FUNCTION_BLOCK FB_System_MVWW_Ablaufsteuerung
VAR_IN_OUT
	Zustand					: ST_System_MVWW_Zustand;
	Stellwert				: ST_System_MVWW_Stellwert;
	Steuerung				: ST_System_MVWW_Steuerung;
END_VAR
VAR_INPUT
	Zustand_Stellventil		: ST_SV_Zustand;
	Zustand_Pumpe			: ST_PU_Zustand;
END_VAR
VAR_OUTPUT
END_VAR
VAR
END_VAR

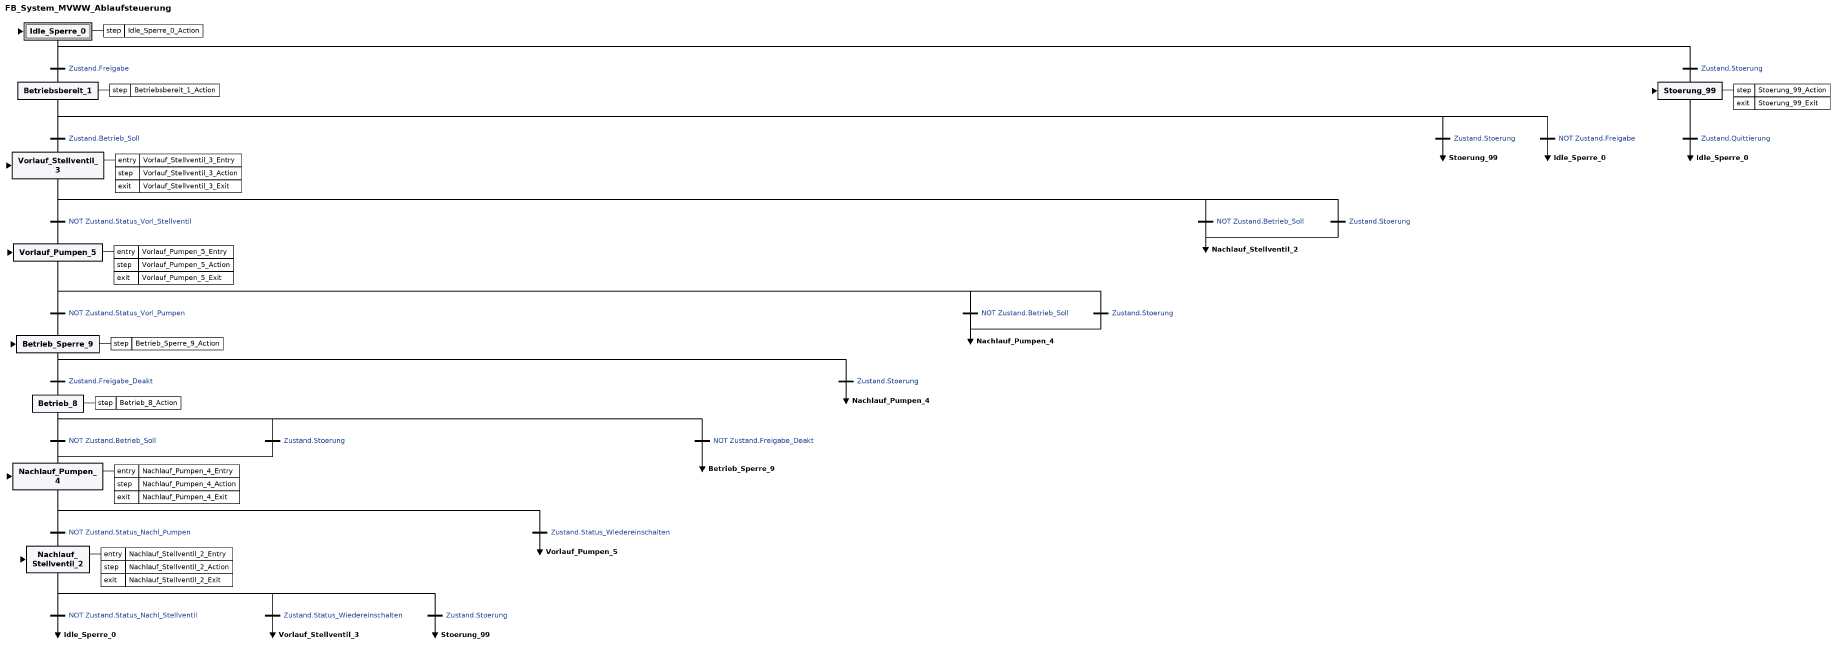
INITIAL_STEP Idle_Sperre_0:
    Idle_Sperre_0_Action(N);  // step action
END_STEP
TRANSITION FROM Idle_Sperre_0 TO Betriebsbereit_1
    := Zustand.Freigabe;
END_TRANSITION
TRANSITION FROM Idle_Sperre_0 TO Stoerung_99
    := Zustand.Stoerung;
END_TRANSITION
STEP Stoerung_99:
    Stoerung_99_Action(N);  // step action
    Stoerung_99_Exit(P0);  // exit action
END_STEP
TRANSITION FROM Stoerung_99 TO Idle_Sperre_0
    := Zustand.Quittierung;
END_TRANSITION
STEP Betriebsbereit_1:
    Betriebsbereit_1_Action(N);  // step action
END_STEP
TRANSITION FROM Betriebsbereit_1 TO Vorlauf_Stellventil_3
    := Zustand.Betrieb_Soll;
END_TRANSITION
TRANSITION FROM Betriebsbereit_1 TO Stoerung_99
    := Zustand.Stoerung;
END_TRANSITION
TRANSITION FROM Betriebsbereit_1 TO Idle_Sperre_0
    := NOT Zustand.Freigabe;
END_TRANSITION
STEP Vorlauf_Stellventil_3:
    Vorlauf_Stellventil_3_Entry(P1);  // entry action
    Vorlauf_Stellventil_3_Action(N);  // step action
    Vorlauf_Stellventil_3_Exit(P0);  // exit action
END_STEP
TRANSITION FROM Vorlauf_Stellventil_3 TO Vorlauf_Pumpen_5
    := NOT Zustand.Status_Vorl_Stellventil;
END_TRANSITION
TRANSITION FROM Vorlauf_Stellventil_3 TO Nachlauf_Stellventil_2
    := NOT Zustand.Betrieb_Soll;
END_TRANSITION
TRANSITION FROM Vorlauf_Stellventil_3 TO Nachlauf_Stellventil_2
    := Zustand.Stoerung;
END_TRANSITION
STEP Vorlauf_Pumpen_5:
    Vorlauf_Pumpen_5_Entry(P1);  // entry action
    Vorlauf_Pumpen_5_Action(N);  // step action
    Vorlauf_Pumpen_5_Exit(P0);  // exit action
END_STEP
TRANSITION FROM Vorlauf_Pumpen_5 TO Betrieb_Sperre_9
    := NOT Zustand.Status_Vorl_Pumpen;
END_TRANSITION
TRANSITION FROM Vorlauf_Pumpen_5 TO Nachlauf_Pumpen_4
    := NOT Zustand.Betrieb_Soll;
END_TRANSITION
TRANSITION FROM Vorlauf_Pumpen_5 TO Nachlauf_Pumpen_4
    := Zustand.Stoerung;
END_TRANSITION
STEP Betrieb_Sperre_9:
    Betrieb_Sperre_9_Action(N);  // step action
END_STEP
TRANSITION FROM Betrieb_Sperre_9 TO Betrieb_8
    := Zustand.Freigabe_Deakt;
END_TRANSITION
TRANSITION FROM Betrieb_Sperre_9 TO Nachlauf_Pumpen_4
    := Zustand.Stoerung;
END_TRANSITION
STEP Betrieb_8:
    Betrieb_8_Action(N);  // step action
END_STEP
TRANSITION FROM Betrieb_8 TO Nachlauf_Pumpen_4
    := NOT Zustand.Betrieb_Soll;
END_TRANSITION
TRANSITION FROM Betrieb_8 TO Nachlauf_Pumpen_4
    := Zustand.Stoerung;
END_TRANSITION
TRANSITION FROM Betrieb_8 TO Betrieb_Sperre_9
    := NOT Zustand.Freigabe_Deakt;
END_TRANSITION
STEP Nachlauf_Pumpen_4:
    Nachlauf_Pumpen_4_Entry(P1);  // entry action
    Nachlauf_Pumpen_4_Action(N);  // step action
    Nachlauf_Pumpen_4_Exit(P0);  // exit action
END_STEP
TRANSITION FROM Nachlauf_Pumpen_4 TO Nachlauf_Stellventil_2
    := NOT Zustand.Status_Nachl_Pumpen;
END_TRANSITION
TRANSITION FROM Nachlauf_Pumpen_4 TO Vorlauf_Pumpen_5
    := Zustand.Status_Wiedereinschalten;
END_TRANSITION
STEP Nachlauf_Stellventil_2:
    Nachlauf_Stellventil_2_Entry(P1);  // entry action
    Nachlauf_Stellventil_2_Action(N);  // step action
    Nachlauf_Stellventil_2_Exit(P0);  // exit action
END_STEP
TRANSITION FROM Nachlauf_Stellventil_2 TO Idle_Sperre_0
    := NOT Zustand.Status_Nachl_Stellventil;
END_TRANSITION
TRANSITION FROM Nachlauf_Stellventil_2 TO Vorlauf_Stellventil_3
    := Zustand.Status_Wiedereinschalten;
END_TRANSITION
TRANSITION FROM Nachlauf_Stellventil_2 TO Stoerung_99
    := Zustand.Stoerung;
END_TRANSITION

ACTION Betrieb_8_Action:
(* Stellwert setzen *)
Stellwert.Anford_Stellventil	:= TRUE;
Stellwert.Anford_Pumpe			:= TRUE;

(* Zustand setzen *)
Zustand.Status					:= E_System_MVWW_Zustand_Status_Betrieb;
END_ACTION

ACTION Betrieb_Sperre_9_Action:
(* Stellwert setzen *)
Stellwert.Anford_Stellventil		:= TRUE;
Stellwert.Anford_Pumpe				:= TRUE;


(* Zustand setzen *)
Zustand.Status						:= E_System_MVWW_Zustand_Status_Betrieb_Sperre;
END_ACTION

ACTION Betriebsbereit_1_Action:
(* Stellwert setzen *)
Stellwert.Anford_Stellventil	:= FALSE;
Stellwert.Anford_Pumpe			:= FALSE;

(* Zustand setzen *)
Zustand.Status			:= E_System_MVWW_Zustand_Status_Betriebsbereit;
END_ACTION

ACTION Idle_Sperre_0_Action:
(* Stellwert setzen *)
Stellwert.Anford_Stellventil		:= FALSE;
Stellwert.Anford_Pumpe				:= FALSE;

(* Zustand setzen *)
Zustand.Status						:= E_System_MVWW_Zustand_Status_Idle_Sperre;

(* Quittierungszustand auf False setzen, damit das System bei einer erneuten Störung nicht direkt wieder angeschaltet wird *)
Steuerung.Quittierung				:= FALSE;
END_ACTION

ACTION Nachlauf_Pumpen_4_Action:
(* Stellwert setzen *)
Stellwert.Anford_Stellventil	:= FALSE;
Stellwert.Anford_Pumpe			:= FALSE;


(* Zustand setzen *)
Zustand.Status						:= E_System_MVWW_Zustand_Status_Nachl_Pumpe;
Zustand.Status_Nachl_Pumpen			:= Zustand_Pumpe.Betrieb OR  Zustand_Pumpe.Status_Nachl;
Zustand.Status_Wiedereinschalten 	:= Zustand.Betrieb_Soll AND Stellwert.Einschalten;
END_ACTION

ACTION Nachlauf_Pumpen_4_Entry:
Zustand.Status_Nachl_Pumpen	:= TRUE;
END_ACTION

ACTION Nachlauf_Pumpen_4_Exit:
Zustand.Status_Nachl_Pumpen	:= FALSE;
END_ACTION

ACTION Nachlauf_Stellventil_2_Action:
(* Stellwert setzen *)
Stellwert.Anford_Stellventil		:= FALSE;
Stellwert.Anford_Pumpe				:= FALSE;

(* Zustand setzen *)
Zustand.Status						:= E_System_MVWW_Zustand_Status_Nachl_Stellventil;
Zustand.Status_Nachl_Stellventil	:= Zustand_Stellventil.Stellung OR Zustand_Stellventil.Stellungwechsel10;
Zustand.Status_Wiedereinschalten 	:= Zustand.Betrieb_Soll AND Stellwert.Einschalten;
END_ACTION

ACTION Nachlauf_Stellventil_2_Entry:
Zustand.Status_Nachl_Stellventil	:= TRUE;
END_ACTION

ACTION Nachlauf_Stellventil_2_Exit:
Zustand.Status_Nachl_Stellventil	:= FALSE;
END_ACTION

ACTION Stoerung_99_Action:
(* Stellwert setzen *)
Stellwert.Anford_Stellventil	:= FALSE;
Stellwert.Anford_Pumpe			:= FALSE;


(* Zustand setzen *)
Zustand.Stoerung				:= TRUE;
Zustand.Status					:= E_System_MVWW_Zustand_Status_Stoerung;
END_ACTION

ACTION Stoerung_99_Exit:
Zustand.Stoerung	:= FALSE;
END_ACTION

ACTION Vorlauf_Pumpen_5_Action:
(* Stellwert setzen *)
Stellwert.Anford_Stellventil		:= TRUE;
Stellwert.Anford_Pumpe				:= TRUE;

(* Zustand setzen *)
Zustand.Status						:= E_System_MVWW_Zustand_Status_Vorl_Pumpe;
Zustand.Status_Vorl_Pumpen			:= NOT(Zustand_Pumpe.Betrieb AND NOT Zustand_Pumpe.Status_Vorl);
END_ACTION

ACTION Vorlauf_Pumpen_5_Entry:
Zustand.Status_Vorl_Pumpen	:= TRUE;
END_ACTION

ACTION Vorlauf_Pumpen_5_Exit:
Zustand.Status_Vorl_Pumpen	:= FALSE;
END_ACTION

ACTION Vorlauf_Stellventil_3_Action:
(* Stellwert setzen *)
Stellwert.Anford_Stellventil		:= TRUE;
Stellwert.Anford_Pumpe				:= FALSE;

(* Zustand setzen *)
Zustand.Status						:= E_System_MVWW_Zustand_Status_Vorl_Stellventil;
Zustand.Status_Vorl_Stellventil		:= NOT(Zustand_Stellventil.Stellung AND NOT Zustand_Stellventil.Stellungwechsel01);
END_ACTION

ACTION Vorlauf_Stellventil_3_Entry:
Zustand.Status_Vorl_Stellventil	:= TRUE;
END_ACTION

ACTION Vorlauf_Stellventil_3_Exit:
Zustand.Status_Vorl_Stellventil	:= FALSE;
END_ACTION

END_FUNCTION_BLOCK

(* stored: Version 1.1.0.1, ProductVersion 3.1.4024.9
   POU FB_System_MVWW_Ablaufsteuerung: Id {9ed8d104-d6db-45e9-bd93-12d661a1d274}, SpecialFunc None
   Action Betrieb_8_Action: Id {157d9962-c420-40d3-8361-1c557d305c3d}
   Action Betrieb_Sperre_9_Action: Id {462a7b58-ec34-40bf-8427-03482d058d96}
   Action Betriebsbereit_1_Action: Id {d5c75d54-587c-44e5-9d28-f86d5f4eb80a}
   Action Idle_Sperre_0_Action: Id {38ab69de-3dbd-42c8-a419-9445a14dc031}
   Action Nachlauf_Pumpen_4_Action: Id {8f8f89be-1848-483e-96cb-fc95fd64ab85}
   Action Nachlauf_Pumpen_4_Entry: Id {e46318dc-5632-4df8-984e-1e2ed6367e15}
   Action Nachlauf_Pumpen_4_Exit: Id {49ec8e2e-07a7-4a30-8082-67e62d610dba}
   Action Nachlauf_Stellventil_2_Action: Id {4b25bdec-d699-41ef-867b-0818bb3bfdef}
   Action Nachlauf_Stellventil_2_Entry: Id {ea08cfaa-45ed-4b78-9d1a-f9e83b212b35}
   Action Nachlauf_Stellventil_2_Exit: Id {e05d72b7-5c14-49b0-9e0a-ae4df71fd592}
   Action Stoerung_99_Action: Id {b2d95903-60f1-4345-a3e7-df288fe4c6a9}
   Action Stoerung_99_Exit: Id {27dcbb93-c3f4-4b98-97c1-10613ba56149}
   Action Vorlauf_Pumpen_5_Action: Id {4d8739ca-fba4-488e-990f-8152c3609b7e}
   Action Vorlauf_Pumpen_5_Entry: Id {c96f0472-6d9b-4c18-940d-d29e0b96e1a0}
   Action Vorlauf_Pumpen_5_Exit: Id {1036af61-69ab-4a4c-8cba-b624e8063a34}
   Action Vorlauf_Stellventil_3_Action: Id {a5715f8a-a6d2-44ae-affa-68cdec0423b2}
   Action Vorlauf_Stellventil_3_Entry: Id {0c22324b-e2f0-49c1-a018-2b4be5f47fff}
   Action Vorlauf_Stellventil_3_Exit: Id {bc242750-66e3-4c20-a758-fd6ec81705d8} *)
